{attribute 'strict'}
TYPE E_RTCCameraInitState :
(
	RTC_INIT_CONNECTION 			:= 0,
	RTC_INIT_CLEAR_BUFFER			:= 10,	
	RTC_INIT_WAIT_FOR_CONFIRMATION	:= 20,
	RTC_INIT_DONE					:= 30
);
END_TYPE

(* stored: Version 1.1.0.1, ProductVersion 3.1.4024.9
   DUT E_RTCCameraInitState: Id {39019f03-aa5f-4b55-98d9-c9d412957118} *)
